FUNCTION_BLOCK XtsTrack EXTENDS CyclicBase IMPLEMENTS I_XtsTrack, I_Initialisable
VAR
	_MyInterface : I_TcIoXtsXpuTrack;
	XtsIoEnvInitialiseState : INT;
	MyPartCount : UDINT;
	Parts : REFERENCE TO ARRAY[1..TcIoXtsEnvironmentParameterList.MaxPartsPerTrack] OF ST_PartInfoItems;
	_TrackLength: LREAL;
	_TrackIsClosed: BOOL;
	_OTCID : OTCID;
	_IsTrackIncludedForDetection : BOOL;
	_NumberOfPartsInTrack : INT;
	_TrackPolarity: Tc3_XTS_Utility.Polarity;
	_IsInitialised : BOOL;
END_VAR

METHOD PUBLIC  Cycle : HRESULT
VAR_INPUT
END_VAR
IF _MyInterface = 0 THEN
	Cycle := -1;
	RETURN;
END_IF

_IsTrackIncludedForDetection := _MyInterface.GetIsIncludedInDetection();
END_METHOD

METHOD Initialise : HRESULT
VAR_INPUT
END_VAR
Initialise := -1;
CASE XtsIoEnvInitialiseState OF
	0:
		IF _MyInterface <> 0 THEN
			XtsIoEnvInitialiseState := 1;
		ELSE
			XtsIoEnvInitialiseState := 999;
		END_IF
	1:
		MyPartCount := _MyInterface.GetPartCount();
		XtsIoEnvInitialiseState := 2;
	2:
		XtsIoEnvInitialiseState := 3;
		Parts REF= _MyInterface.GetPartInfoItems();
		
	3:
		IF _MyInterface.P_IsInitialized THEN
			_TrackLength := _MyInterface.GetLength();
			_TrackIsClosed := _MyInterface.GetIsClosed();
			_TrackPolarity := _MyInterface.GetPolarity();
			_NumberOfPartsInTrack := TO_INT(_MyInterface.GetPartCount());
			XtsIoEnvInitialiseState := 4;
		END_IF
	4:
		Initialise := 0;
		_IsInitialised := TRUE;
END_CASE
END_METHOD

PROPERTY Initialised : BOOL
GET
Initialised := _IsInitialised;
END_GET
END_PROPERTY

PROPERTY MyOTCID : OTCID
GET
MyOTCID := _OTCID;
END_GET
SET
_OTCID := MyOTCID;
END_SET
END_PROPERTY

PROPERTY MyXtsIoEnvInterface : I_TcIoXtsXpuTrack
GET
MyXtsIoEnvInterface := _MyInterface;
END_GET
SET
_MyInterface := MyXtsIoEnvInterface;
END_SET
END_PROPERTY

PROPERTY NumberOfPartsInTrack : INT
GET
NumberOfPartsInTrack := _NumberOfPartsInTrack;
END_GET
END_PROPERTY

METHOD RemoveFromDetection : BOOL
VAR_INPUT
END_VAR
RemoveFromDetection := _MyInterface.SetIsIncludedInDetection(False);
END_METHOD

METHOD SetForDetection : BOOL
VAR_INPUT
END_VAR
SetForDetection := _MyInterface.SetIsIncludedInDetection(TRUE);
END_METHOD

PROPERTY TrackLength : MC_Lreal
GET
TrackLength := _MyInterface.GetLength();
END_GET
END_PROPERTY

END_FUNCTION_BLOCK

(* stored: Version 1.1.0.1
   POU XtsTrack: Id {0ed646c8-24dd-40d8-b451-d6e6a88b90d3}, SpecialFunc None
   Folder Commands: Id {32cad632-fbd4-445a-b2c2-d8eaa1f5efa0}
   Folder Settings: Id {b0f2811b-01c3-4263-ae13-de05f982e5bb}
   Folder Status: Id {574d2b11-115b-44b2-972f-d3d465c1b172}
   Method Cycle: Id {753f4845-bb32-46bd-9afe-0c535a6bb9c5}
   Method Initialise: Id {b15a1974-ae41-45a0-b8ce-e38654aa0808}
   Property Initialised: Id {339e97b4-50a8-4342-a310-e8536eaede2f}
   Get Get: Id {76068666-6775-4f24-bbb9-a431dc2f8a5e}
   Property MyOTCID: Id {d34cfe46-c497-4e94-b74d-f99a6000b358}
   Get Get: Id {855c0947-7cfe-4f24-8259-2331fd728b0d}
   Set Set: Id {52d396c9-aa72-4a6c-b0f5-3d8704d35aca}
   Property MyXtsIoEnvInterface: Id {de406d6a-fb33-4758-a1bb-071b44e09534}
   Get Get: Id {29c07896-dd74-4eb2-b4f6-620c540248e5}
   Set Set: Id {efa5de65-cd69-47bf-b917-2b3471279c8e}
   Property NumberOfPartsInTrack: Id {4227d870-553b-4fcb-8516-6ae7f6500149}
   Get Get: Id {47e7e73c-f2f4-4613-aa92-016379f2eda9}
   Method RemoveFromDetection: Id {19fc9c17-6e83-4583-8661-ca0f3d7fbe00}
   Method SetForDetection: Id {2a4c4b2d-af72-4d4f-81aa-5409f825db3c}
   Property TrackLength: Id {f63b8800-afc4-4a64-a819-7bbd5ce82fd4}
   Get Get: Id {8c76ee9b-64b1-4933-b3fe-20fbe5dcfddc} *)
